FUNCTION_BLOCK SubSystemButtonWidget
VAR_INPUT
    color : StatusColor;
    hideColor : BOOL := FALSE;
END_VAR
VAR_IN_OUT
    activeTab : INT;
END_VAR
VAR_OUTPUT
    name : STRING;
    thisTab : INT;
    colorVisible : BOOL;
    
    activated : BOOL;
    notActivated : BOOL;
    
    isNotGreen : BOOL;
    isNotRed : BOOL;
    isNotBlue : BOOL;
    isNotOrange : BOOL;
    isNotGray : BOOL;
END_VAR
VAR
    do_activate : BOOL;
END_VAR


IF do_activate THEN
    activeTab := thisTab;
    do_activate := FALSE;
END_IF

activated := activeTab = thisTab;
notActivated := NOT activated;

isNotRed    := color.bg <> Colors.RED;
isNotBlue   := color.bg <> Colors.BLUE;
isNotOrange := color.bg <> Colors.ORANGE;
isNotGray   := color.bg <> Colors.GRAY;
isNotGreen  := color.bg <> Colors.GREEN;

METHOD FB_init : BOOL
VAR_INPUT
	bInitRetains : BOOL; // if TRUE, the retain variables are initialized (warm start / cold start)
	bInCopyCode : BOOL;  // if TRUE, the instance afterwards gets moved into the copy code (online change)
    n : STRING;
    tab : INT;
END_VAR
name := n;
thisTab := tab;
END_METHOD

END_FUNCTION_BLOCK

(* stored: Version 1.1.0.1, ProductVersion 3.1.4018.2
   POU SubSystemButtonWidget: Id {3ea39677-d223-4ec2-8260-2c9f826c9076}, SpecialFunc None
   Method FB_init: Id {a74b41b6-342c-48e2-86ee-f84f6fd1861c} *)
